// SIMATIC S7-200 project (STEP 7-Micro/WIN), CPU 224 REL 02.01

ORGANIZATION_BLOCK PRINCIPAL:OB1
TITLE=CONTROL_AJUSTABLE - JEVG
BEGIN
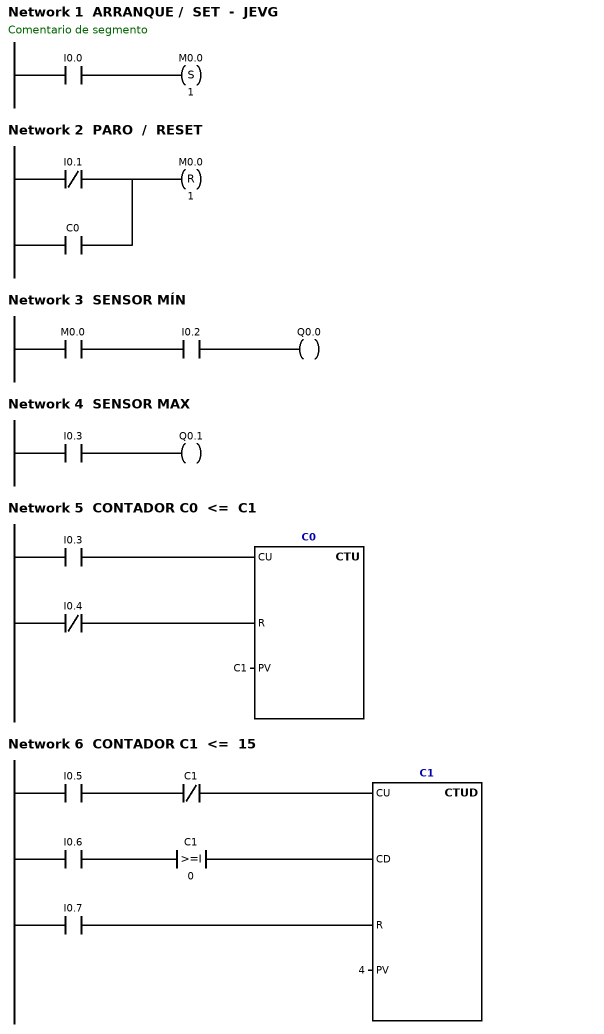
Network 1 // ARRANQUE /  SET  -  JEVG
// Comentario de segmento
LD     I0.0
S      M0.0, 1
Network 2 // PARO  /  RESET
LDN    I0.1
O      C0
R      M0.0, 1
Network 3 // SENSOR MÍN
LD     M0.0
A      I0.2
=      Q0.0
Network 4 // SENSOR MAX 
LD     I0.3
=      Q0.1
Network 5 // CONTADOR C0  <=  C1
LD     I0.3
LDN    I0.4
CTU    C0, C1
Network 6 // CONTADOR C1  <=  15
LD     I0.5
AN     C1
LD     I0.6
AW>=   C1, 0
LD     I0.7
CTUD   C1, 4
END_ORGANIZATION_BLOCK
